FUNCTION_BLOCK ABSTRACT SuspendedToRunningProgramTransition EXTENDS ProgramTransition

{attribute 'monitoring' := 'call'}
{attribute 'OPC.UA.DA.Property' := '1'}
{attribute 'OPC.UA.DA.Access' := '1'}
PROPERTY FINAL Cause : STRING
GET
Cause := 'Resume';
END_GET
END_PROPERTY

{attribute 'monitoring' := 'call'}
{attribute 'OPC.UA.DA.Property' := '1'}
{attribute 'OPC.UA.DA.Access' := '1'}
PROPERTY FINAL FromState : STRING
GET
FromState := 'Suspended';
END_GET
END_PROPERTY

{attribute 'monitoring' := 'call'}
{attribute 'OPC.UA.DA.Property' := '1'}
{attribute 'OPC.UA.DA.Access' := '1'}
PROPERTY FINAL Name : STRING
GET
Name := 'SuspendedToRunning';
END_GET
END_PROPERTY

{attribute 'monitoring' := 'call'}
{attribute 'OPC.UA.DA.Property' := '1'}
{attribute 'OPC.UA.DA.Access' := '1'}
PROPERTY FINAL ToState : STRING
GET
ToState := 'Running';
END_GET
END_PROPERTY

END_FUNCTION_BLOCK

(* stored: Version 1.1.0.1
   POU SuspendedToRunningProgramTransition: Id {73940194-7ad8-4c7d-a7e2-da1428f97644}, SpecialFunc None
   Property Cause: Id {ec67baad-38fa-4640-8208-d6128403e7e1}
   Get Get: Id {e08ff649-ce46-45f2-9356-6276d8c10e23}
   Property FromState: Id {d1f509d5-af93-4d5e-8ccd-7894ed258be1}
   Get Get: Id {570c370a-360d-44d6-b150-88b41d7add70}
   Property Name: Id {c921389e-abd5-45b8-8f55-61d3bcc6517d}
   Get Get: Id {ed24db42-7c6b-4ead-b497-3d0ad090ef8a}
   Property ToState: Id {400fb345-b0a6-442f-8b22-729b539e3211}
   Get Get: Id {a0edc4d5-eb6b-4a88-87ad-1896bee5c5bc} *)
